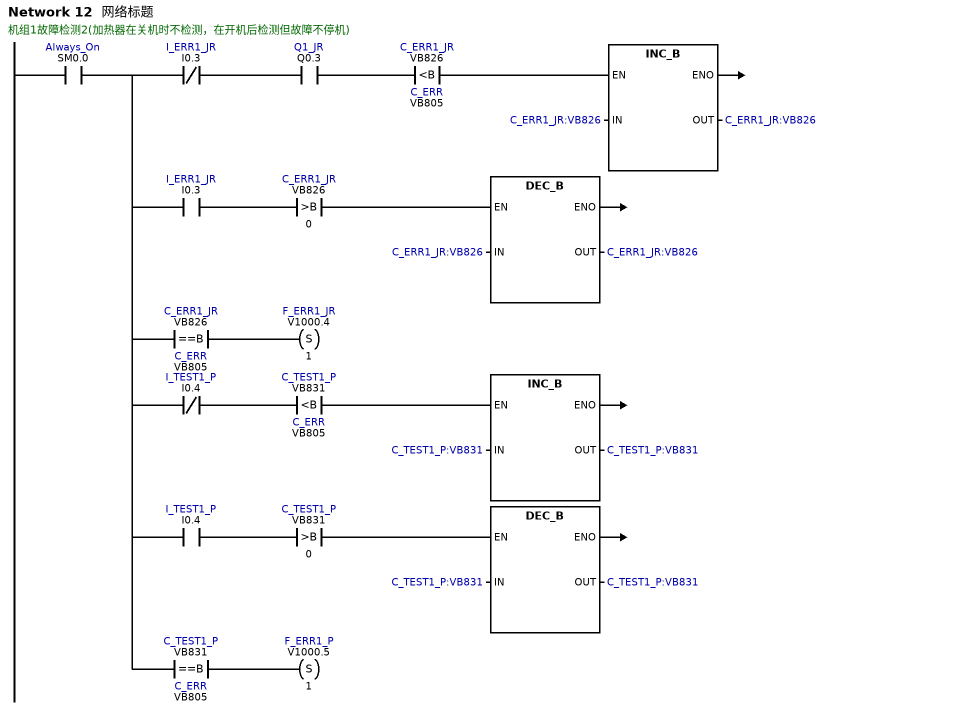
[picture p24: SBR3 networks 12-12]
Network 12 // 网络标题
// 机组1故障检测2(加热器在关机时不检测，在开机后检测但故障不停机)
LD     Always_On:SM0.0
LPS
AN     I_ERR1_JR:I0.3
A      Q1_JR:Q0.3
AB<    C_ERR1_JR:VB826, C_ERR:VB805
INCB   C_ERR1_JR:VB826
LRD
A      I_ERR1_JR:I0.3
AB>    C_ERR1_JR:VB826, 0
DECB   C_ERR1_JR:VB826
LRD
AB=    C_ERR1_JR:VB826, C_ERR:VB805
S      F_ERR1_JR:V1000.4, 1
LRD
AN     I_TEST1_P:I0.4
AB<    C_TEST1_P:VB831, C_ERR:VB805
INCB   C_TEST1_P:VB831
LRD
A      I_TEST1_P:I0.4
AB>    C_TEST1_P:VB831, 0
DECB   C_TEST1_P:VB831
LPP
AB=    C_TEST1_P:VB831, C_ERR:VB805
S      F_ERR1_P:V1000.5, 1
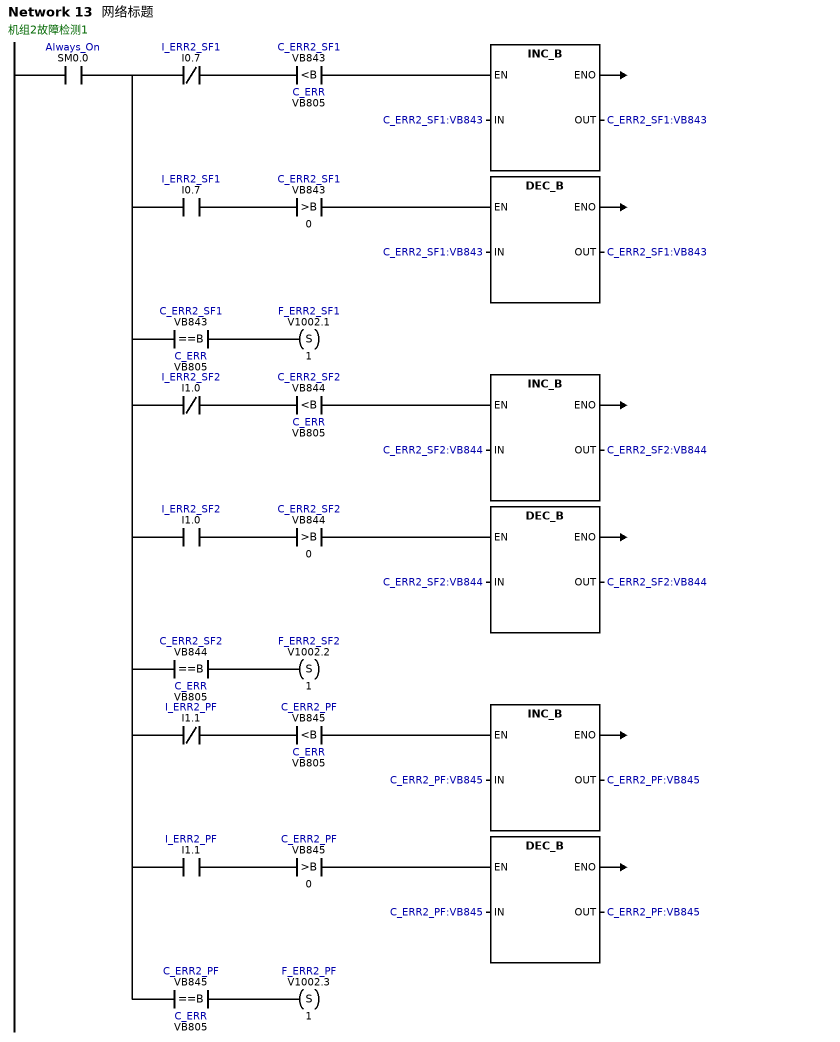
Network 13 // 网络标题
// 机组2故障检测1
LD     Always_On:SM0.0
LPS
AN     I_ERR2_SF1:I0.7
AB<    C_ERR2_SF1:VB843, C_ERR:VB805
INCB   C_ERR2_SF1:VB843
LRD
A      I_ERR2_SF1:I0.7
AB>    C_ERR2_SF1:VB843, 0
DECB   C_ERR2_SF1:VB843
LRD
AB=    C_ERR2_SF1:VB843, C_ERR:VB805
S      F_ERR2_SF1:V1002.1, 1
LRD
AN     I_ERR2_SF2:I1.0
AB<    C_ERR2_SF2:VB844, C_ERR:VB805
INCB   C_ERR2_SF2:VB844
LRD
A      I_ERR2_SF2:I1.0
AB>    C_ERR2_SF2:VB844, 0
DECB   C_ERR2_SF2:VB844
LRD
AB=    C_ERR2_SF2:VB844, C_ERR:VB805
S      F_ERR2_SF2:V1002.2, 1
LRD
AN     I_ERR2_PF:I1.1
AB<    C_ERR2_PF:VB845, C_ERR:VB805
INCB   C_ERR2_PF:VB845
LRD
A      I_ERR2_PF:I1.1
AB>    C_ERR2_PF:VB845, 0
DECB   C_ERR2_PF:VB845
LPP
AB=    C_ERR2_PF:VB845, C_ERR:VB805
S      F_ERR2_PF:V1002.3, 1
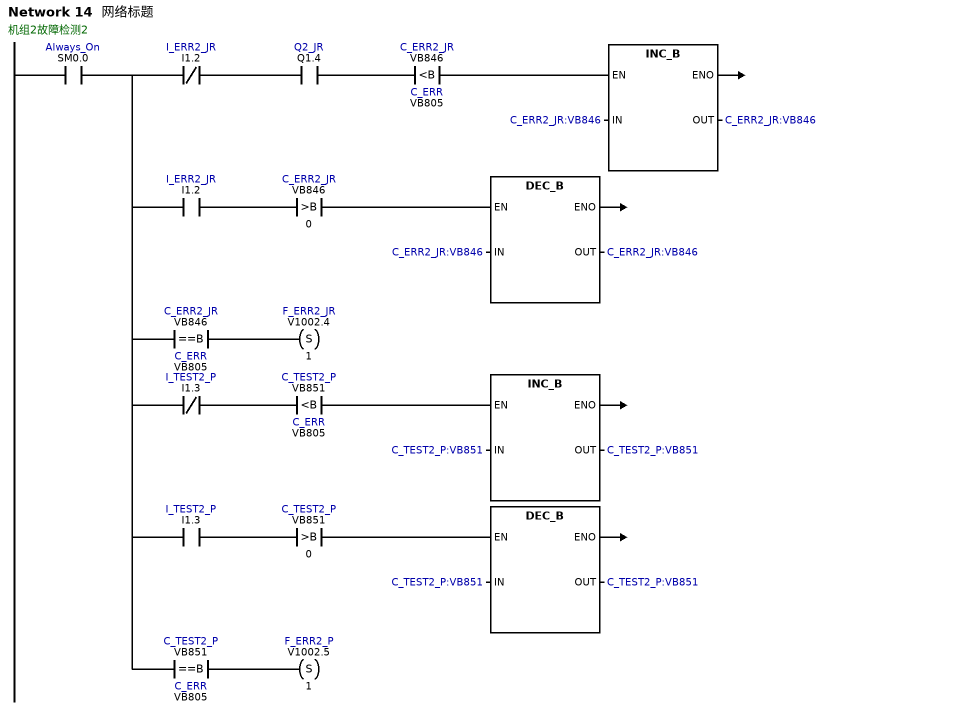
Network 14 // 网络标题
// 机组2故障检测2
LD     Always_On:SM0.0
LPS
AN     I_ERR2_JR:I1.2
A      Q2_JR:Q1.4
AB<    C_ERR2_JR:VB846, C_ERR:VB805
INCB   C_ERR2_JR:VB846
LRD
A      I_ERR2_JR:I1.2
AB>    C_ERR2_JR:VB846, 0
DECB   C_ERR2_JR:VB846
LRD
AB=    C_ERR2_JR:VB846, C_ERR:VB805
S      F_ERR2_JR:V1002.4, 1
LRD
AN     I_TEST2_P:I1.3
AB<    C_TEST2_P:VB851, C_ERR:VB805
INCB   C_TEST2_P:VB851
LRD
A      I_TEST2_P:I1.3
AB>    C_TEST2_P:VB851, 0
DECB   C_TEST2_P:VB851
LPP
AB=    C_TEST2_P:VB851, C_ERR:VB805
S      F_ERR2_P:V1002.5, 1
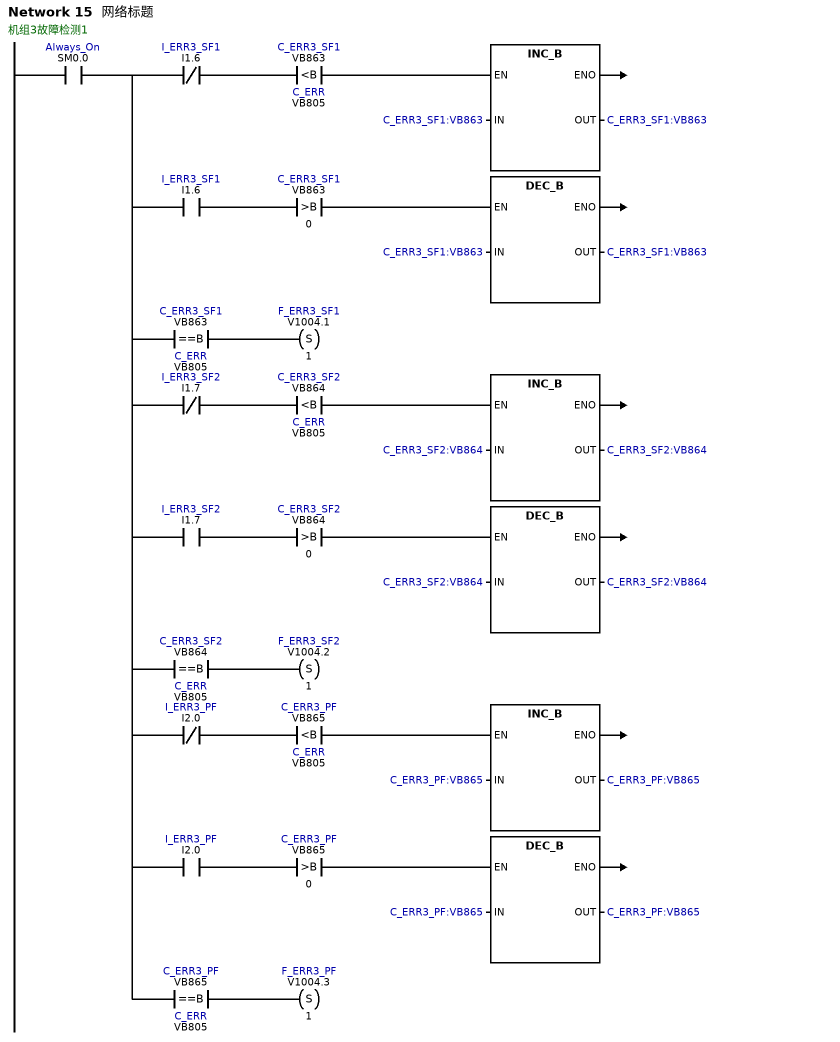
Network 15 // 网络标题
// 机组3故障检测1
LD     Always_On:SM0.0
LPS
AN     I_ERR3_SF1:I1.6
AB<    C_ERR3_SF1:VB863, C_ERR:VB805
INCB   C_ERR3_SF1:VB863
LRD
A      I_ERR3_SF1:I1.6
AB>    C_ERR3_SF1:VB863, 0
DECB   C_ERR3_SF1:VB863
LRD
AB=    C_ERR3_SF1:VB863, C_ERR:VB805
S      F_ERR3_SF1:V1004.1, 1
LRD
AN     I_ERR3_SF2:I1.7
AB<    C_ERR3_SF2:VB864, C_ERR:VB805
INCB   C_ERR3_SF2:VB864
LRD
A      I_ERR3_SF2:I1.7
AB>    C_ERR3_SF2:VB864, 0
DECB   C_ERR3_SF2:VB864
LRD
AB=    C_ERR3_SF2:VB864, C_ERR:VB805
S      F_ERR3_SF2:V1004.2, 1
LRD
AN     I_ERR3_PF:I2.0
AB<    C_ERR3_PF:VB865, C_ERR:VB805
INCB   C_ERR3_PF:VB865
LRD
A      I_ERR3_PF:I2.0
AB>    C_ERR3_PF:VB865, 0
DECB   C_ERR3_PF:VB865
LPP
AB=    C_ERR3_PF:VB865, C_ERR:VB805
S      F_ERR3_PF:V1004.3, 1
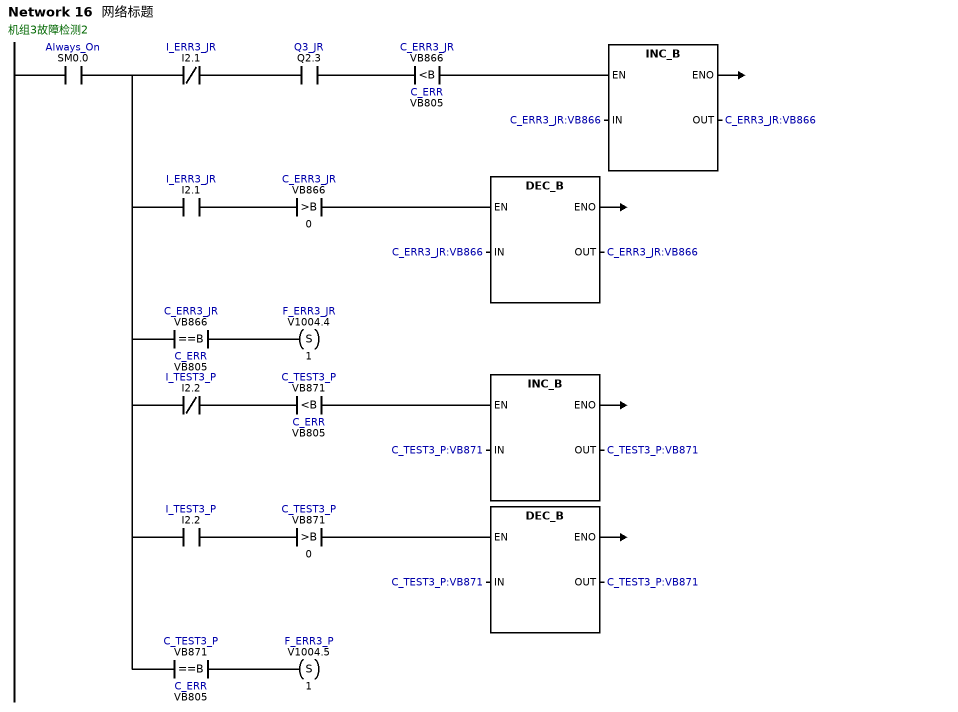
Network 16 // 网络标题
// 机组3故障检测2
LD     Always_On:SM0.0
LPS
AN     I_ERR3_JR:I2.1
A      Q3_JR:Q2.3
AB<    C_ERR3_JR:VB866, C_ERR:VB805
INCB   C_ERR3_JR:VB866
LRD
A      I_ERR3_JR:I2.1
AB>    C_ERR3_JR:VB866, 0
DECB   C_ERR3_JR:VB866
LRD
AB=    C_ERR3_JR:VB866, C_ERR:VB805
S      F_ERR3_JR:V1004.4, 1
LRD
AN     I_TEST3_P:I2.2
AB<    C_TEST3_P:VB871, C_ERR:VB805
INCB   C_TEST3_P:VB871
LRD
A      I_TEST3_P:I2.2
AB>    C_TEST3_P:VB871, 0
DECB   C_TEST3_P:VB871
LPP
AB=    C_TEST3_P:VB871, C_ERR:VB805
S      F_ERR3_P:V1004.5, 1
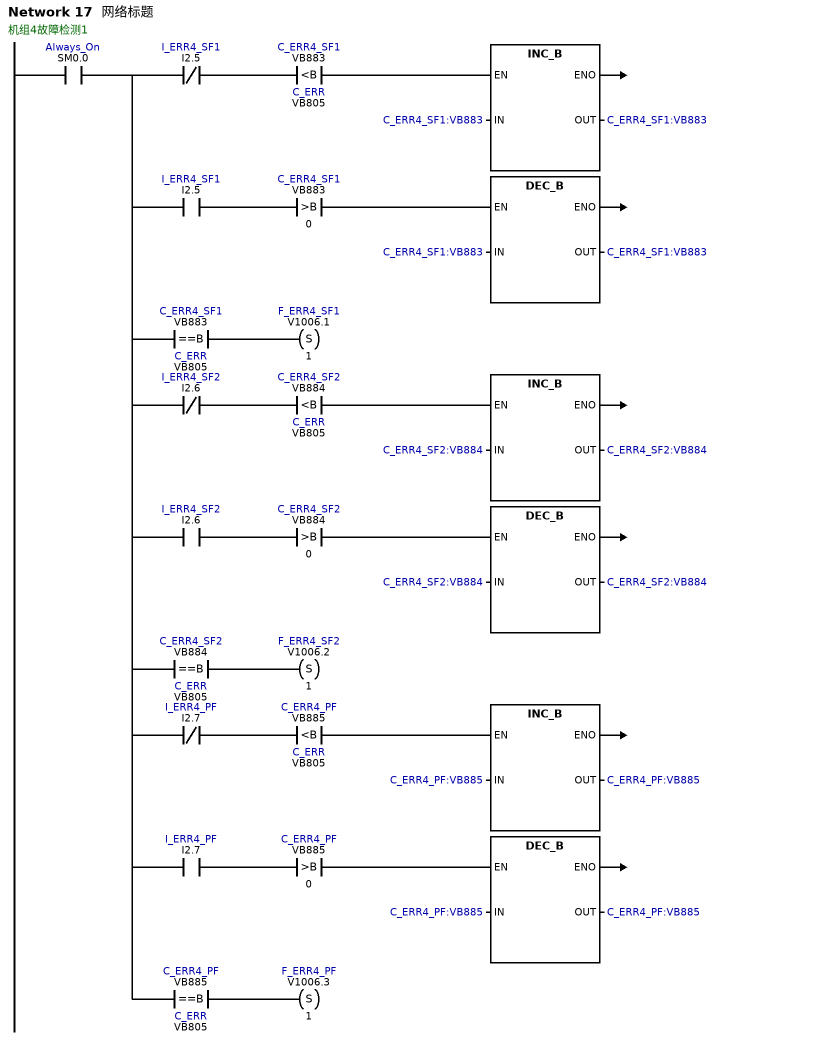
Network 17 // 网络标题
// 机组4故障检测1
LD     Always_On:SM0.0
LPS
AN     I_ERR4_SF1:I2.5
AB<    C_ERR4_SF1:VB883, C_ERR:VB805
INCB   C_ERR4_SF1:VB883
LRD
A      I_ERR4_SF1:I2.5
AB>    C_ERR4_SF1:VB883, 0
DECB   C_ERR4_SF1:VB883
LRD
AB=    C_ERR4_SF1:VB883, C_ERR:VB805
S      F_ERR4_SF1:V1006.1, 1
LRD
AN     I_ERR4_SF2:I2.6
AB<    C_ERR4_SF2:VB884, C_ERR:VB805
INCB   C_ERR4_SF2:VB884
LRD
A      I_ERR4_SF2:I2.6
AB>    C_ERR4_SF2:VB884, 0
DECB   C_ERR4_SF2:VB884
LRD
AB=    C_ERR4_SF2:VB884, C_ERR:VB805
S      F_ERR4_SF2:V1006.2, 1
LRD
AN     I_ERR4_PF:I2.7
AB<    C_ERR4_PF:VB885, C_ERR:VB805
INCB   C_ERR4_PF:VB885
LRD
A      I_ERR4_PF:I2.7
AB>    C_ERR4_PF:VB885, 0
DECB   C_ERR4_PF:VB885
LPP
AB=    C_ERR4_PF:VB885, C_ERR:VB805
S      F_ERR4_PF:V1006.3, 1
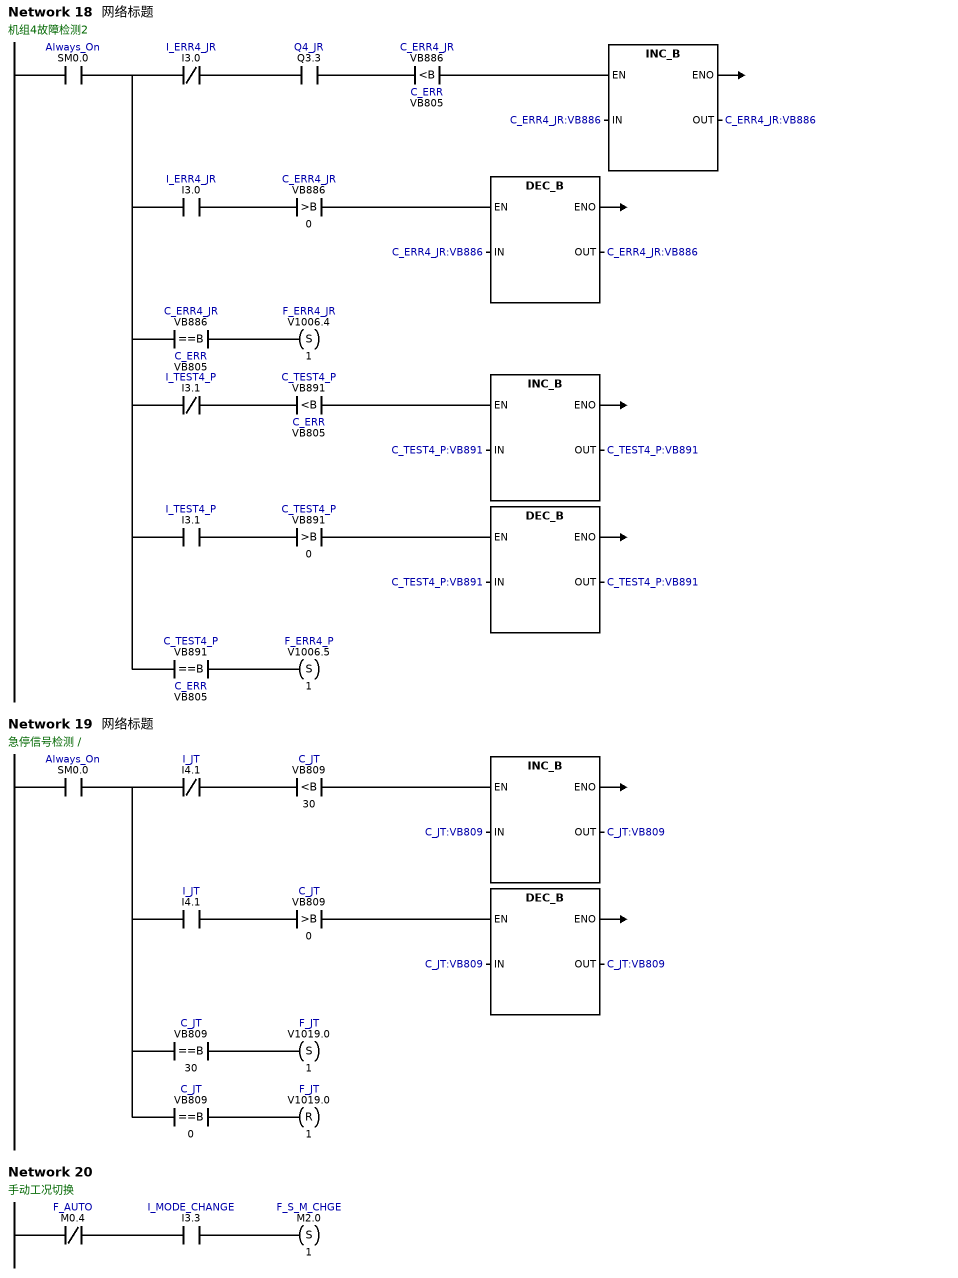
Network 18 // 网络标题
// 机组4故障检测2
LD     Always_On:SM0.0
LPS
AN     I_ERR4_JR:I3.0
A      Q4_JR:Q3.3
AB<    C_ERR4_JR:VB886, C_ERR:VB805
INCB   C_ERR4_JR:VB886
LRD
A      I_ERR4_JR:I3.0
AB>    C_ERR4_JR:VB886, 0
DECB   C_ERR4_JR:VB886
LRD
AB=    C_ERR4_JR:VB886, C_ERR:VB805
S      F_ERR4_JR:V1006.4, 1
LRD
AN     I_TEST4_P:I3.1
AB<    C_TEST4_P:VB891, C_ERR:VB805
INCB   C_TEST4_P:VB891
LRD
A      I_TEST4_P:I3.1
AB>    C_TEST4_P:VB891, 0
DECB   C_TEST4_P:VB891
LPP
AB=    C_TEST4_P:VB891, C_ERR:VB805
S      F_ERR4_P:V1006.5, 1
Network 19 // 网络标题
// 急停信号检测
// 
LD     Always_On:SM0.0
LPS
AN     I_JT:I4.1
AB<    C_JT:VB809, 30
INCB   C_JT:VB809
LRD
A      I_JT:I4.1
AB>    C_JT:VB809, 0
DECB   C_JT:VB809
LRD
AB=    C_JT:VB809, 30
S      F_JT:V1019.0, 1
LPP
AB=    C_JT:VB809, 0
R      F_JT:V1019.0, 1
Network 20
// 手动工况切换
LDN    F_AUTO:M0.4
A      I_MODE_CHANGE:I3.3
S      F_S_M_CHGE:M2.0, 1
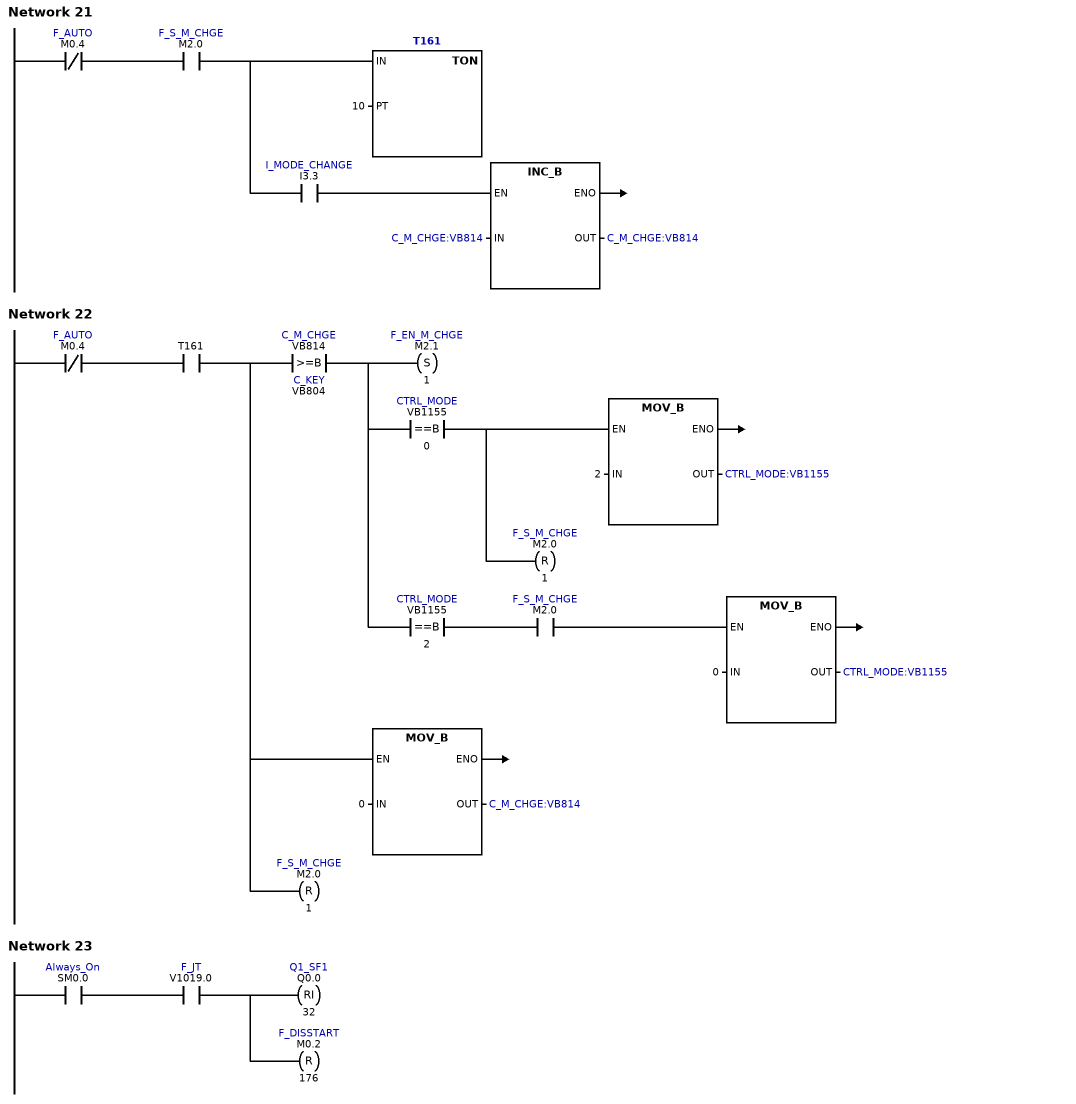
Network 21
LDN    F_AUTO:M0.4
A      F_S_M_CHGE:M2.0
TON    T161, 10
A      I_MODE_CHANGE:I3.3
INCB   C_M_CHGE:VB814
Network 22
LDN    F_AUTO:M0.4
A      T161
LPS
AB>=   C_M_CHGE:VB814, C_KEY:VB804
LPS
S      F_EN_M_CHGE:M2.1, 1
AB=    CTRL_MODE:VB1155, 0
MOVB   2, CTRL_MODE:VB1155
R      F_S_M_CHGE:M2.0, 1
LPP
AB=    CTRL_MODE:VB1155, 2
A      F_S_M_CHGE:M2.0
MOVB   0, CTRL_MODE:VB1155
LPP
MOVB   0, C_M_CHGE:VB814
R      F_S_M_CHGE:M2.0, 1
Network 23
LD     Always_On:SM0.0
A      F_JT:V1019.0
RI     Q1_SF1:Q0.0, 32
R      F_DISSTART:M0.2, 176
END_SUBROUTINE_BLOCK

// SBR4: protected block, not included

SUBROUTINE_BLOCK 参数设定:SBR5
TITLE=
VAR
TEMP_W:WORD;	// LW0 
TEMP_W1:WORD;	// LW2 
TEMP_W2:WORD;	// LW4 
END_VAR
BEGIN
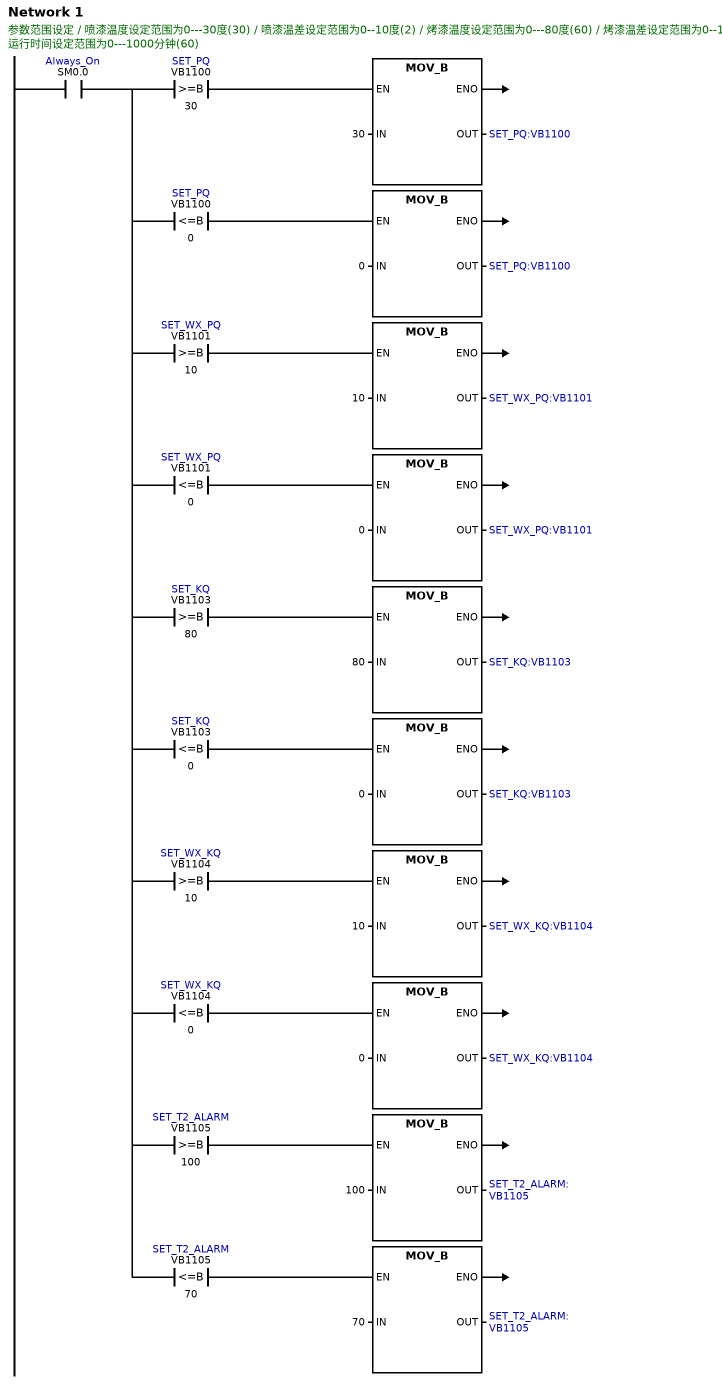
Network 1
// 参数范围设定
// 喷漆温度设定范围为0---30度(30)
// 喷漆温差设定范围为0--10度(2)
// 烤漆温度设定范围为0---80度(60)
// 烤漆温差设定范围为0--10度(2)
// T2超温保护温度设定范围为70---100度(85)
// 运行时间设定范围为0---1000分钟(60)
LD     Always_On:SM0.0
LPS
AB>=   SET_PQ:VB1100, 30
MOVB   30, SET_PQ:VB1100
LRD
AB<=   SET_PQ:VB1100, 0
MOVB   0, SET_PQ:VB1100
LRD
AB>=   SET_WX_PQ:VB1101, 10
MOVB   10, SET_WX_PQ:VB1101
LRD
AB<=   SET_WX_PQ:VB1101, 0
MOVB   0, SET_WX_PQ:VB1101
LRD
AB>=   SET_KQ:VB1103, 80
MOVB   80, SET_KQ:VB1103
LRD
AB<=   SET_KQ:VB1103, 0
MOVB   0, SET_KQ:VB1103
LRD
AB>=   SET_WX_KQ:VB1104, 10
MOVB   10, SET_WX_KQ:VB1104
LRD
AB<=   SET_WX_KQ:VB1104, 0
MOVB   0, SET_WX_KQ:VB1104
LRD
AB>=   SET_T2_ALARM:VB1105, 100
MOVB   100, SET_T2_ALARM:VB1105
LPP
AB<=   SET_T2_ALARM:VB1105, 70
MOVB   70, SET_T2_ALARM:VB1105
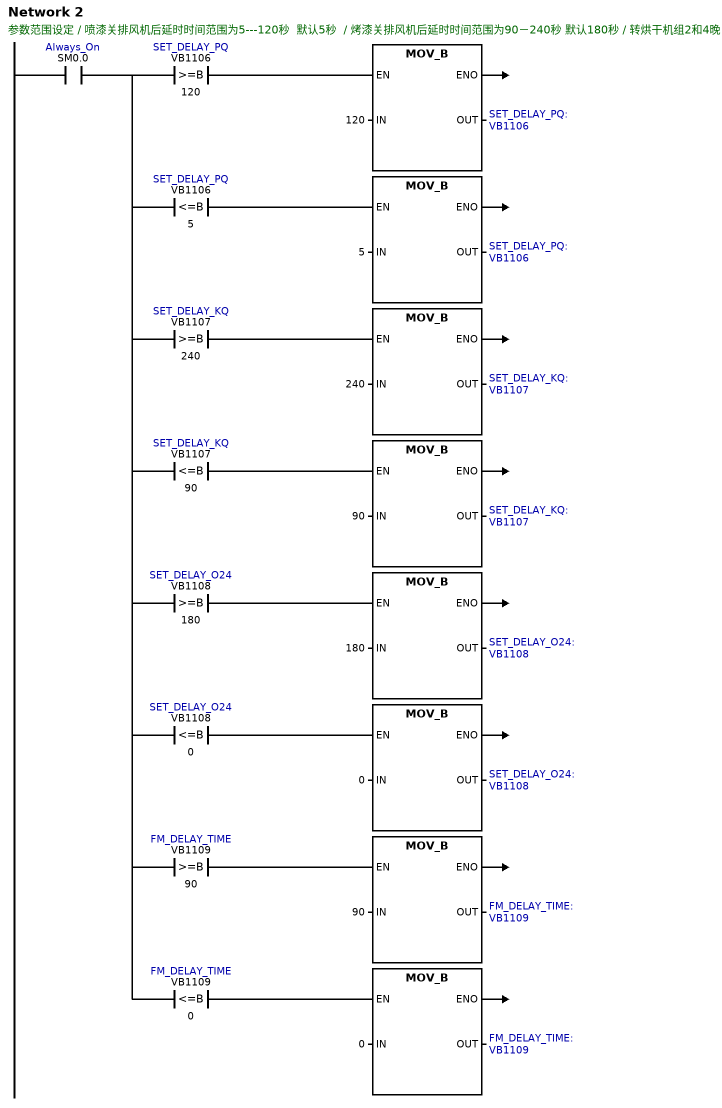
Network 2
// 参数范围设定
// 喷漆关排风机后延时时间范围为5---120秒  默认5秒 
// 烤漆关排风机后延时时间范围为90－240秒 默认180秒
// 转烘干机组2和4晚关延时时间为0－180秒   默认30秒
LD     Always_On:SM0.0
LPS
AB>=   SET_DELAY_PQ:VB1106, 120
MOVB   120, SET_DELAY_PQ:VB1106
LRD
AB<=   SET_DELAY_PQ:VB1106, 5
MOVB   5, SET_DELAY_PQ:VB1106
LRD
AB>=   SET_DELAY_KQ:VB1107, 240
MOVB   240, SET_DELAY_KQ:VB1107
LRD
AB<=   SET_DELAY_KQ:VB1107, 90
MOVB   90, SET_DELAY_KQ:VB1107
LRD
AB>=   SET_DELAY_O24:VB1108, 180
MOVB   180, SET_DELAY_O24:VB1108
LRD
AB<=   SET_DELAY_O24:VB1108, 0
MOVB   0, SET_DELAY_O24:VB1108
LRD
AB>=   FM_DELAY_TIME:VB1109, 90
MOVB   90, FM_DELAY_TIME:VB1109
LPP
AB<=   FM_DELAY_TIME:VB1109, 0
MOVB   0, FM_DELAY_TIME:VB1109
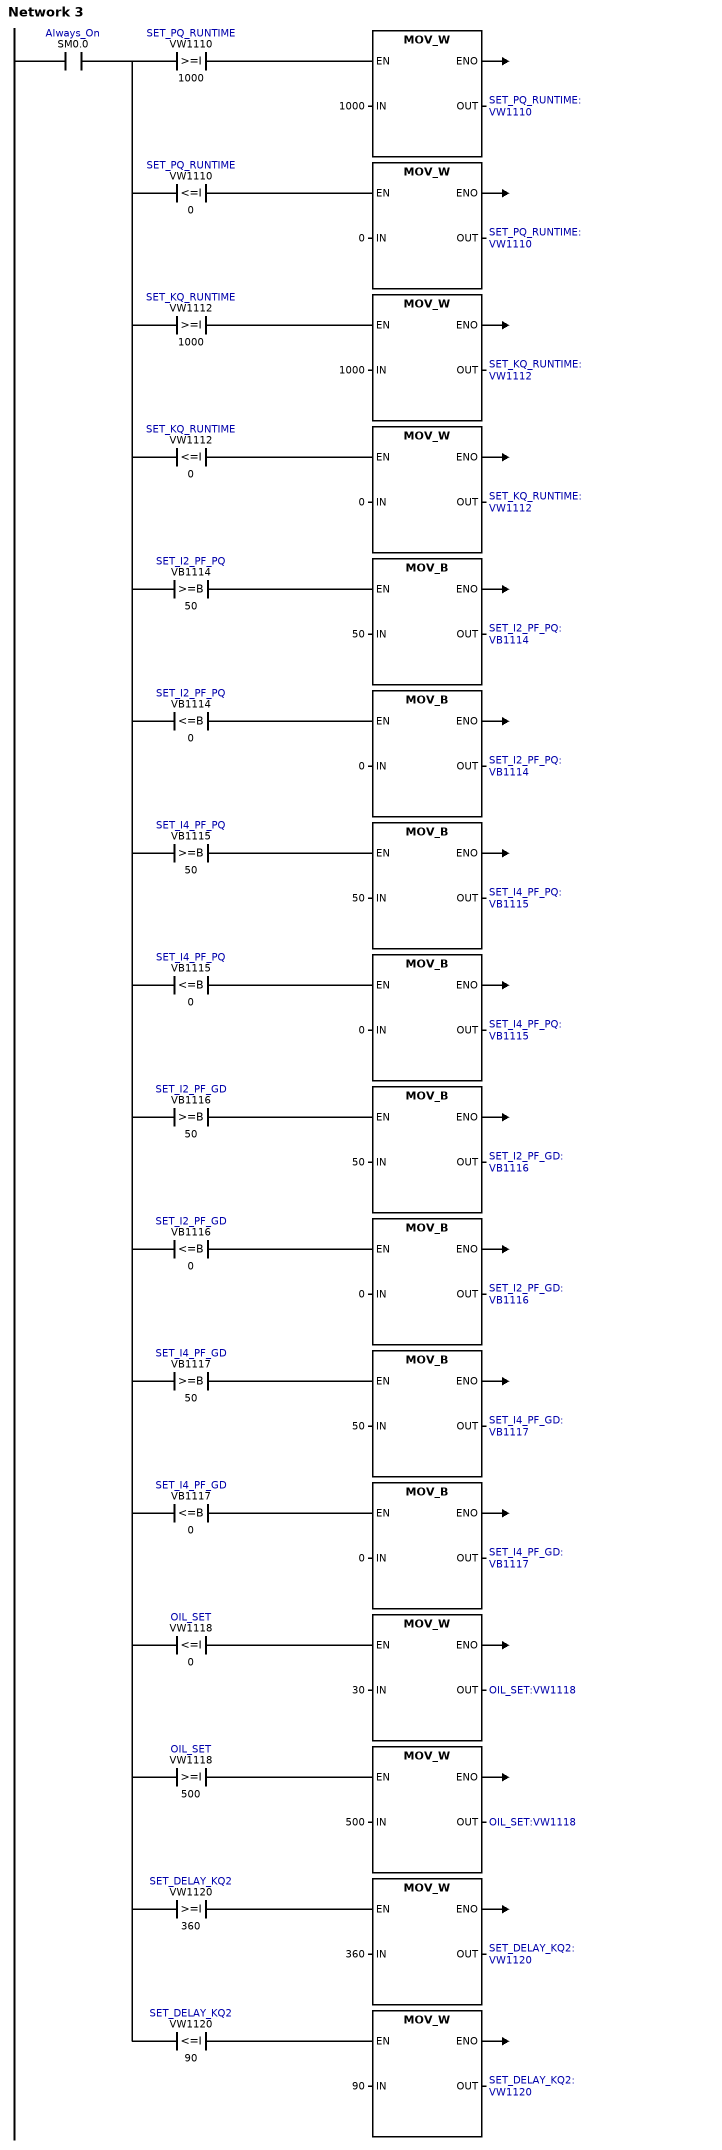
Network 3
LD     Always_On:SM0.0
LPS
AW>=   SET_PQ_RUNTIME:VW1110, 1000
MOVW   1000, SET_PQ_RUNTIME:VW1110
LRD
AW<=   SET_PQ_RUNTIME:VW1110, 0
MOVW   0, SET_PQ_RUNTIME:VW1110
LRD
AW>=   SET_KQ_RUNTIME:VW1112, 1000
MOVW   1000, SET_KQ_RUNTIME:VW1112
LRD
AW<=   SET_KQ_RUNTIME:VW1112, 0
MOVW   0, SET_KQ_RUNTIME:VW1112
LRD
AB>=   SET_I2_PF_PQ:VB1114, 50
MOVB   50, SET_I2_PF_PQ:VB1114
LRD
AB<=   SET_I2_PF_PQ:VB1114, 0
MOVB   0, SET_I2_PF_PQ:VB1114
LRD
AB>=   SET_I4_PF_PQ:VB1115, 50
MOVB   50, SET_I4_PF_PQ:VB1115
LRD
AB<=   SET_I4_PF_PQ:VB1115, 0
MOVB   0, SET_I4_PF_PQ:VB1115
LRD
AB>=   SET_I2_PF_GD:VB1116, 50
MOVB   50, SET_I2_PF_GD:VB1116
LRD
AB<=   SET_I2_PF_GD:VB1116, 0
MOVB   0, SET_I2_PF_GD:VB1116
LRD
AB>=   SET_I4_PF_GD:VB1117, 50
MOVB   50, SET_I4_PF_GD:VB1117
LRD
AB<=   SET_I4_PF_GD:VB1117, 0
MOVB   0, SET_I4_PF_GD:VB1117
LRD
AW<=   OIL_SET:VW1118, 0
MOVW   30, OIL_SET:VW1118
LRD
AW>=   OIL_SET:VW1118, 500
MOVW   500, OIL_SET:VW1118
LRD
AW>=   SET_DELAY_KQ2:VW1120, 360
MOVW   360, SET_DELAY_KQ2:VW1120
LPP
AW<=   SET_DELAY_KQ2:VW1120, 90
MOVW   90, SET_DELAY_KQ2:VW1120
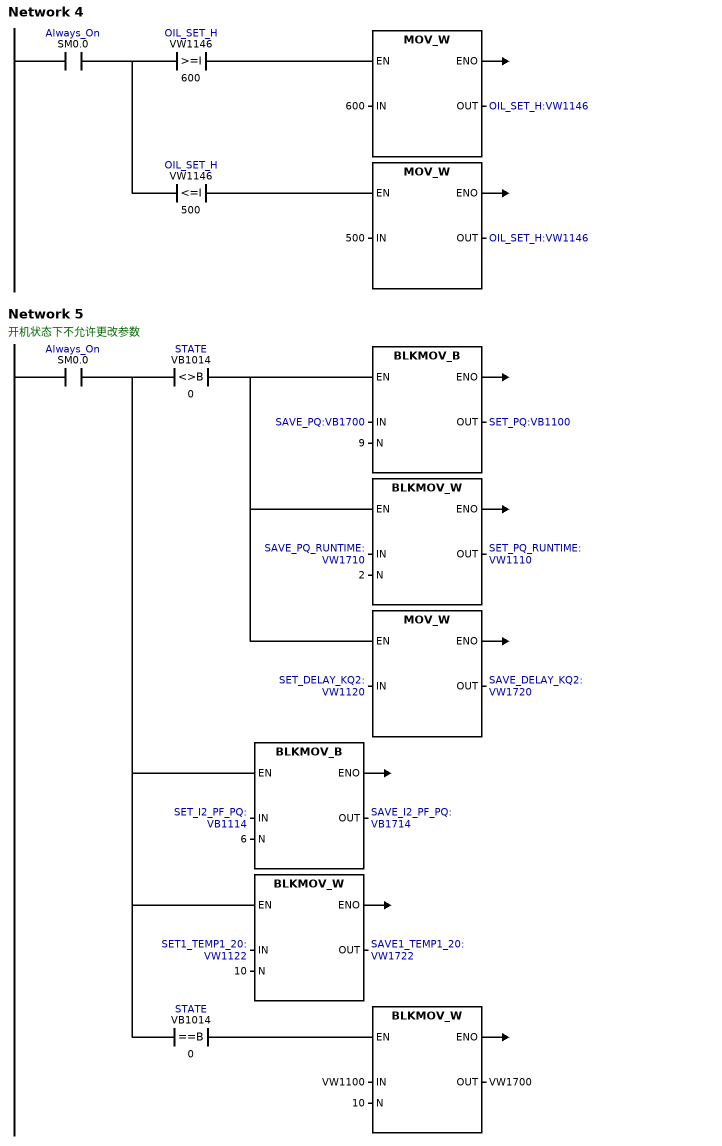
Network 4
LD     Always_On:SM0.0
LPS
AW>=   OIL_SET_H:VW1146, 600
MOVW   600, OIL_SET_H:VW1146
LPP
AW<=   OIL_SET_H:VW1146, 500
MOVW   500, OIL_SET_H:VW1146
Network 5
// 开机状态下不允许更改参数
LD     Always_On:SM0.0
LPS
AB<>   STATE:VB1014, 0
BMB    SAVE_PQ:VB1700, SET_PQ:VB1100, 9
BMW    SAVE_PQ_RUNTIME:VW1710, SET_PQ_RUNTIME:VW1110, 2
MOVW   SET_DELAY_KQ2:VW1120, SAVE_DELAY_KQ2:VW1720
LPP
BMB    SET_I2_PF_PQ:VB1114, SAVE_I2_PF_PQ:VB1714, 6
BMW    SET1_TEMP1_20:VW1122, SAVE1_TEMP1_20:VW1722, 10
AB=    STATE:VB1014, 0
BMW    VW1100, VW1700, 10
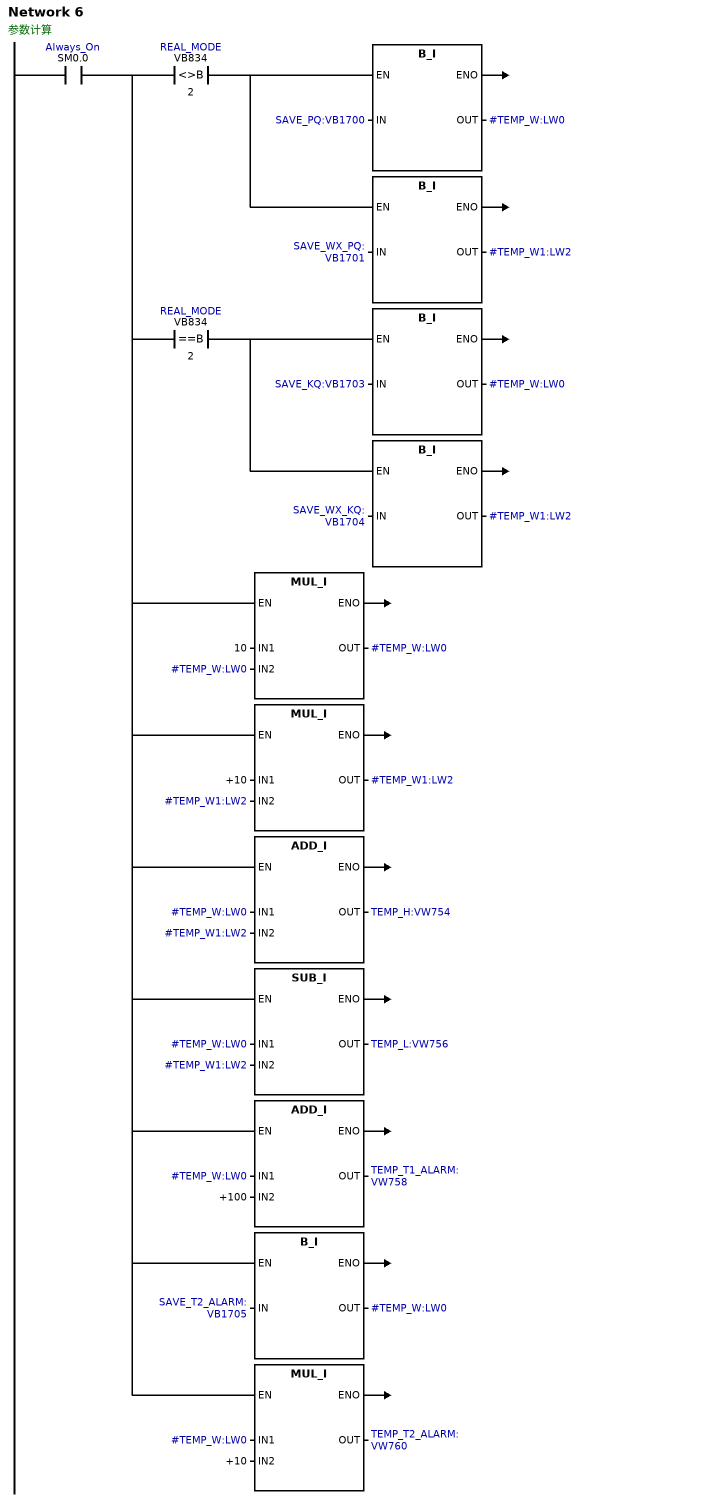
Network 6
// 参数计算
LD     Always_On:SM0.0
LPS
AB<>   REAL_MODE:VB834, 2
BTI    SAVE_PQ:VB1700, #TEMP_W:LW0
BTI    SAVE_WX_PQ:VB1701, #TEMP_W1:LW2
LRD
AB=    REAL_MODE:VB834, 2
BTI    SAVE_KQ:VB1703, #TEMP_W:LW0
BTI    SAVE_WX_KQ:VB1704, #TEMP_W1:LW2
LPP
*I     10, #TEMP_W:LW0
*I     +10, #TEMP_W1:LW2
MOVW   #TEMP_W:LW0, TEMP_H:VW754
+I     #TEMP_W1:LW2, TEMP_H:VW754
MOVW   #TEMP_W:LW0, TEMP_L:VW756
-I     #TEMP_W1:LW2, TEMP_L:VW756
MOVW   #TEMP_W:LW0, TEMP_T1_ALARM:VW758
+I     +100, TEMP_T1_ALARM:VW758
BTI    SAVE_T2_ALARM:VB1705, #TEMP_W:LW0
MOVW   #TEMP_W:LW0, TEMP_T2_ALARM:VW760
*I     +10, TEMP_T2_ALARM:VW760
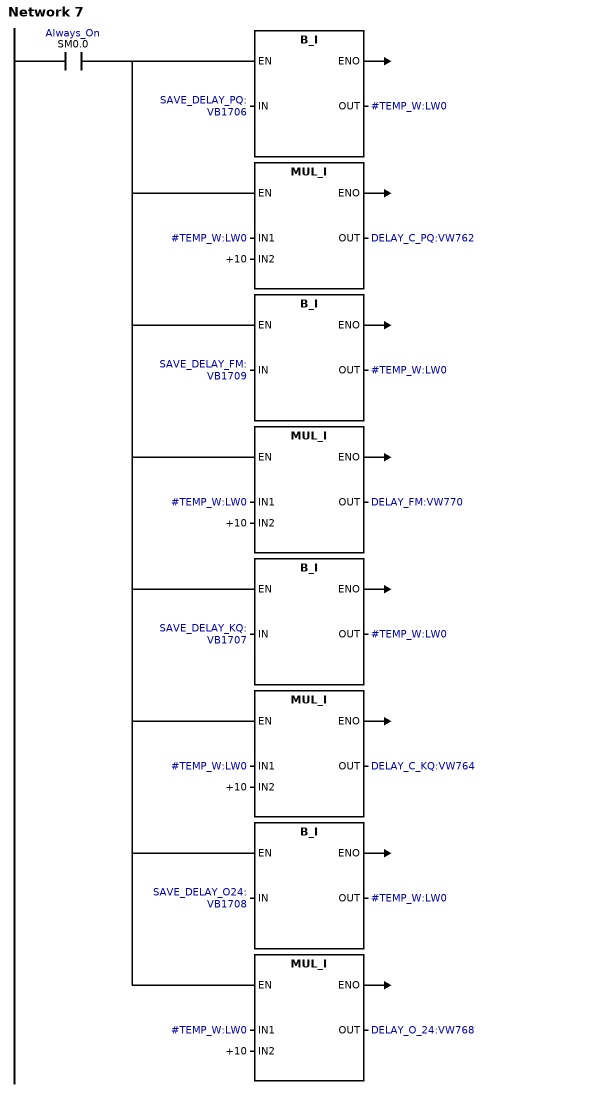
Network 7
LD     Always_On:SM0.0
BTI    SAVE_DELAY_PQ:VB1706, #TEMP_W:LW0
MOVW   #TEMP_W:LW0, DELAY_C_PQ:VW762
*I     +10, DELAY_C_PQ:VW762
BTI    SAVE_DELAY_FM:VB1709, #TEMP_W:LW0
MOVW   #TEMP_W:LW0, DELAY_FM:VW770
*I     +10, DELAY_FM:VW770
BTI    SAVE_DELAY_KQ:VB1707, #TEMP_W:LW0
MOVW   #TEMP_W:LW0, DELAY_C_KQ:VW764
*I     +10, DELAY_C_KQ:VW764
BTI    SAVE_DELAY_O24:VB1708, #TEMP_W:LW0
MOVW   #TEMP_W:LW0, DELAY_O_24:VW768
*I     +10, DELAY_O_24:VW768
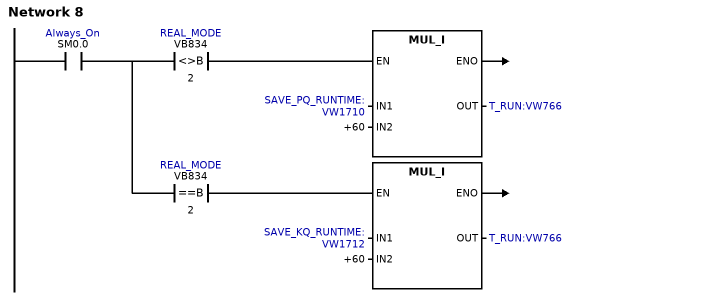
Network 8
LD     Always_On:SM0.0
LPS
AB<>   REAL_MODE:VB834, 2
MOVW   SAVE_PQ_RUNTIME:VW1710, T_RUN:VW766
*I     +60, T_RUN:VW766
LPP
AB=    REAL_MODE:VB834, 2
MOVW   SAVE_KQ_RUNTIME:VW1712, T_RUN:VW766
*I     +60, T_RUN:VW766
END_SUBROUTINE_BLOCK

SUBROUTINE_BLOCK 温度采样:SBR6
TITLE=
VAR_INPUT
ADDRESS:DWORD;	// LD0 
IN:WORD;	// LW4 
IN_TEMP:WORD;	// LW6 
F_SET:BOOL;	// L8.0 
END_VAR
VAR_OUTPUT
OUT:WORD;	// LW9 
AVERAGE:WORD;	// LW11 
OUT_TEMP:WORD;	// LW13 
END_VAR
VAR
MAX:WORD;	// LW15 
MIN:WORD;	// LW17 
TEMP_B:BYTE;	// LB19 
TEMP_W:WORD;	// LW20 
TEMP_DW:DWORD;	// LD22 
SUM:DWORD;	// LD26 
PP1:DWORD;	// LD30 
PP2:DWORD;	// LD34 
TEMP_W2:WORD;	// LW38 
AC_TEMP:DWORD;	// LD40 
END_VAR
BEGIN
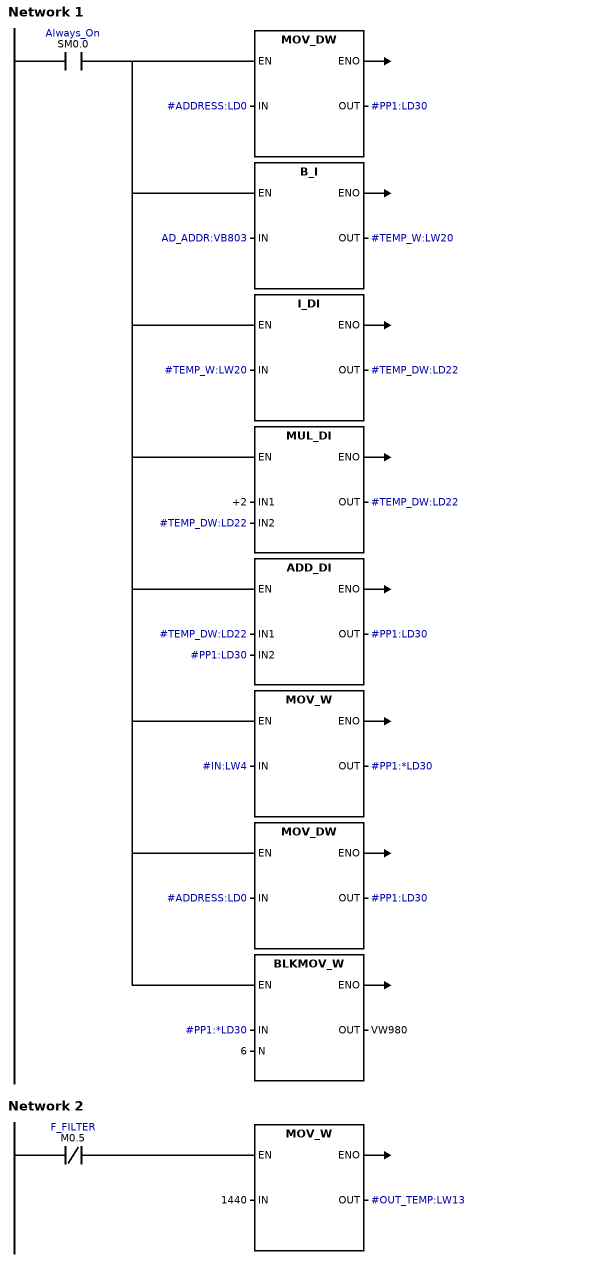
Network 1
LD     Always_On:SM0.0
MOVD   #ADDRESS:LD0, #PP1:LD30
BTI    AD_ADDR:VB803, #TEMP_W:LW20
ITD    #TEMP_W:LW20, #TEMP_DW:LD22
*D     +2, #TEMP_DW:LD22
+D     #TEMP_DW:LD22, #PP1:LD30
MOVW   #IN:LW4, *#PP1:LD30
MOVD   #ADDRESS:LD0, #PP1:LD30
BMW    *#PP1:LD30, VW980, 6
Network 2
LDN    F_FILTER:M0.5
MOVW   1440, #OUT_TEMP:LW13
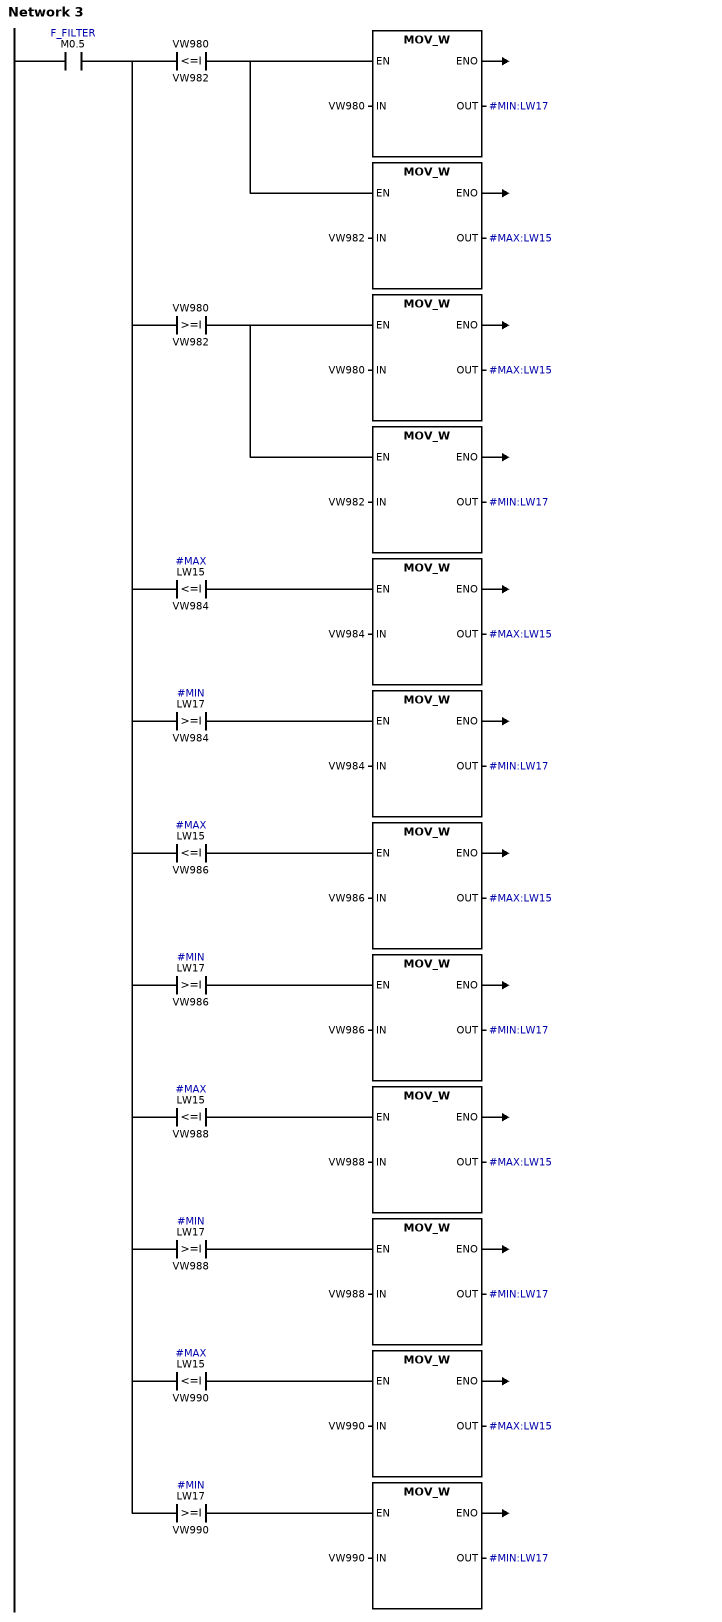
Network 3
LD     F_FILTER:M0.5
LPS
AW<=   VW980, VW982
MOVW   VW980, #MIN:LW17
MOVW   VW982, #MAX:LW15
LRD
AW>=   VW980, VW982
MOVW   VW980, #MAX:LW15
MOVW   VW982, #MIN:LW17
LPP
LPS
AW<=   #MAX:LW15, VW984
MOVW   VW984, #MAX:LW15
LRD
AW>=   #MIN:LW17, VW984
MOVW   VW984, #MIN:LW17
LRD
AW<=   #MAX:LW15, VW986
MOVW   VW986, #MAX:LW15
LRD
AW>=   #MIN:LW17, VW986
MOVW   VW986, #MIN:LW17
LRD
AW<=   #MAX:LW15, VW988
MOVW   VW988, #MAX:LW15
LRD
AW>=   #MIN:LW17, VW988
MOVW   VW988, #MIN:LW17
LRD
AW<=   #MAX:LW15, VW990
MOVW   VW990, #MAX:LW15
LPP
AW>=   #MIN:LW17, VW990
MOVW   VW990, #MIN:LW17
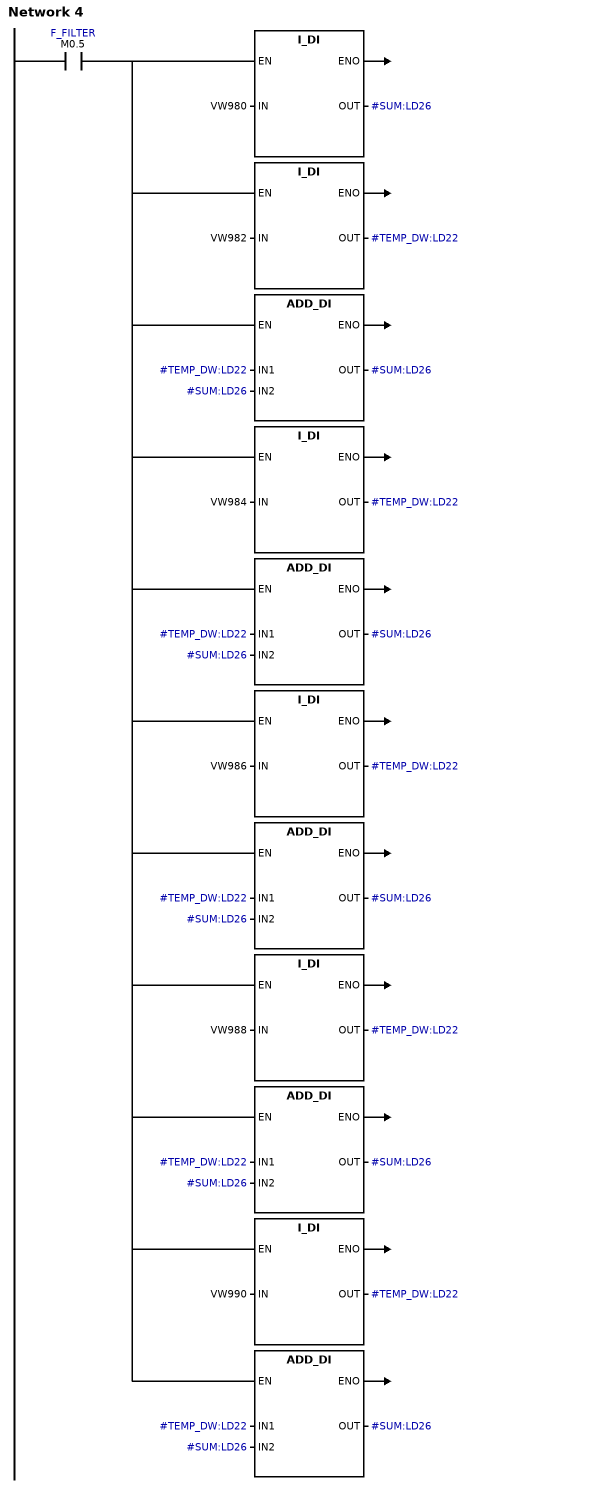
Network 4
LD     F_FILTER:M0.5
ITD    VW980, #SUM:LD26
ITD    VW982, #TEMP_DW:LD22
+D     #TEMP_DW:LD22, #SUM:LD26
ITD    VW984, #TEMP_DW:LD22
+D     #TEMP_DW:LD22, #SUM:LD26
ITD    VW986, #TEMP_DW:LD22
+D     #TEMP_DW:LD22, #SUM:LD26
ITD    VW988, #TEMP_DW:LD22
+D     #TEMP_DW:LD22, #SUM:LD26
ITD    VW990, #TEMP_DW:LD22
+D     #TEMP_DW:LD22, #SUM:LD26
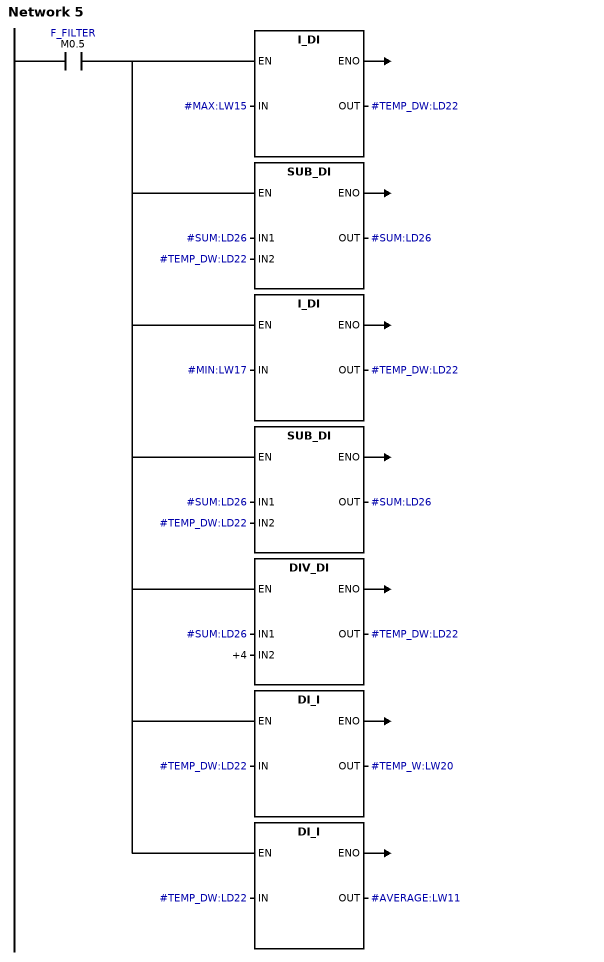
Network 5
LD     F_FILTER:M0.5
ITD    #MAX:LW15, #TEMP_DW:LD22
-D     #TEMP_DW:LD22, #SUM:LD26
ITD    #MIN:LW17, #TEMP_DW:LD22
-D     #TEMP_DW:LD22, #SUM:LD26
MOVD   #SUM:LD26, #TEMP_DW:LD22
/D     +4, #TEMP_DW:LD22
DTI    #TEMP_DW:LD22, #TEMP_W:LW20
DTI    #TEMP_DW:LD22, #AVERAGE:LW11
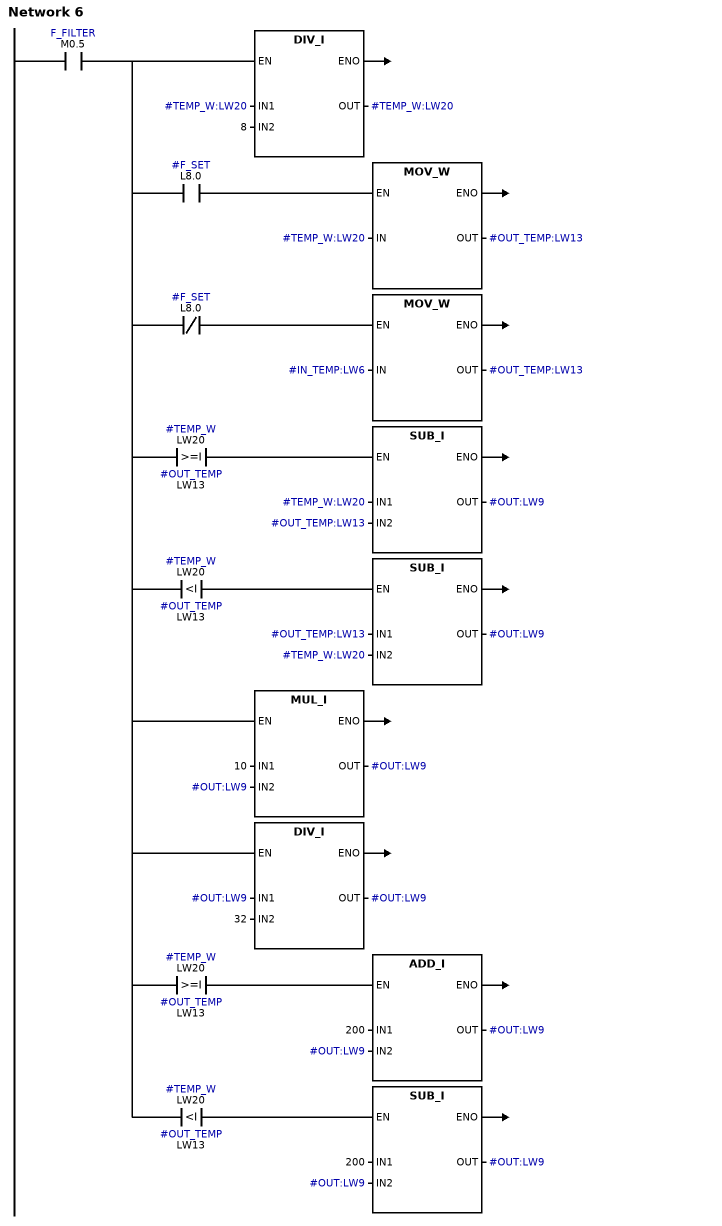
Network 6
LD     F_FILTER:M0.5
LPS
/I     8, #TEMP_W:LW20
A      #F_SET:L8.0
MOVW   #TEMP_W:LW20, #OUT_TEMP:LW13
LRD
AN     #F_SET:L8.0
MOVW   #IN_TEMP:LW6, #OUT_TEMP:LW13
LRD
AW>=   #TEMP_W:LW20, #OUT_TEMP:LW13
MOVW   #TEMP_W:LW20, #OUT:LW9
-I     #OUT_TEMP:LW13, #OUT:LW9
LRD
AW<    #TEMP_W:LW20, #OUT_TEMP:LW13
MOVW   #OUT_TEMP:LW13, #OUT:LW9
-I     #TEMP_W:LW20, #OUT:LW9
LRD
*I     10, #OUT:LW9
LRD
/I     32, #OUT:LW9
LRD
AW>=   #TEMP_W:LW20, #OUT_TEMP:LW13
+I     200, #OUT:LW9
LPP
AW<    #TEMP_W:LW20, #OUT_TEMP:LW13
INVW   #OUT:LW9
INCW   #OUT:LW9
+I     200, #OUT:LW9
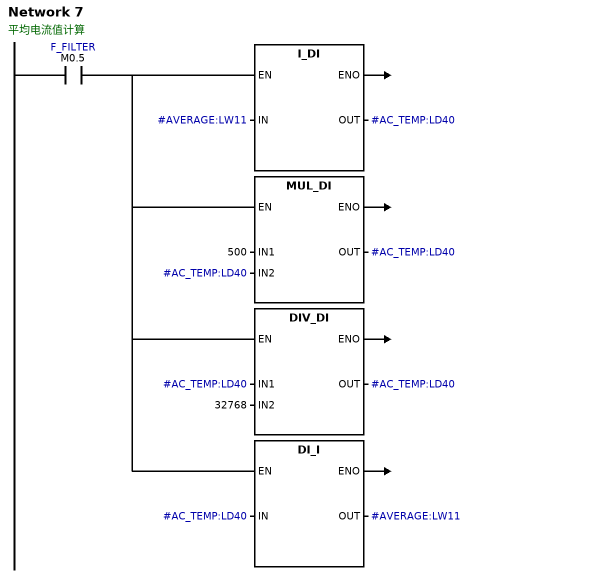
Network 7
// 平均电流值计算
LD     F_FILTER:M0.5
ITD    #AVERAGE:LW11, #AC_TEMP:LD40
*D     500, #AC_TEMP:LD40
/D     32768, #AC_TEMP:LD40
DTI    #AC_TEMP:LD40, #AVERAGE:LW11
END_SUBROUTINE_BLOCK

SUBROUTINE_BLOCK 启动停止控制:SBR7
TITLE=
BEGIN
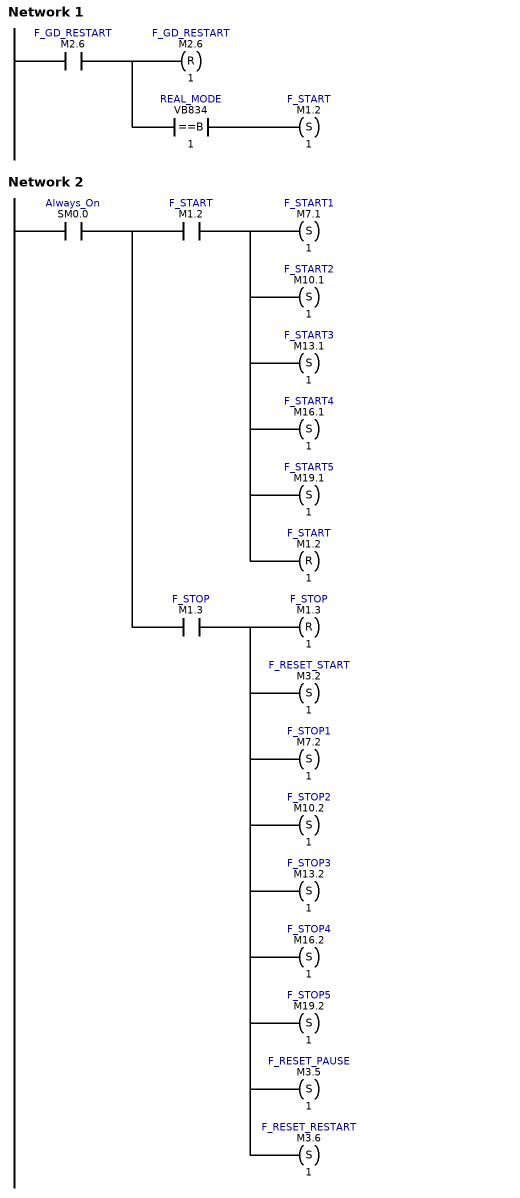
Network 1
LD     F_GD_RESTART:M2.6
R      F_GD_RESTART:M2.6, 1
AB=    REAL_MODE:VB834, 1
S      F_START:M1.2, 1
Network 2
LD     Always_On:SM0.0
LPS
A      F_START:M1.2
S      F_START1:M7.1, 1
S      F_START2:M10.1, 1
S      F_START3:M13.1, 1
S      F_START4:M16.1, 1
S      F_START5:M19.1, 1
R      F_START:M1.2, 1
LPP
A      F_STOP:M1.3
R      F_STOP:M1.3, 1
S      F_RESET_START:M3.2, 1
S      F_STOP1:M7.2, 1
S      F_STOP2:M10.2, 1
S      F_STOP3:M13.2, 1
S      F_STOP4:M16.2, 1
S      F_STOP5:M19.2, 1
S      F_RESET_PAUSE:M3.5, 1
S      F_RESET_RESTART:M3.6, 1
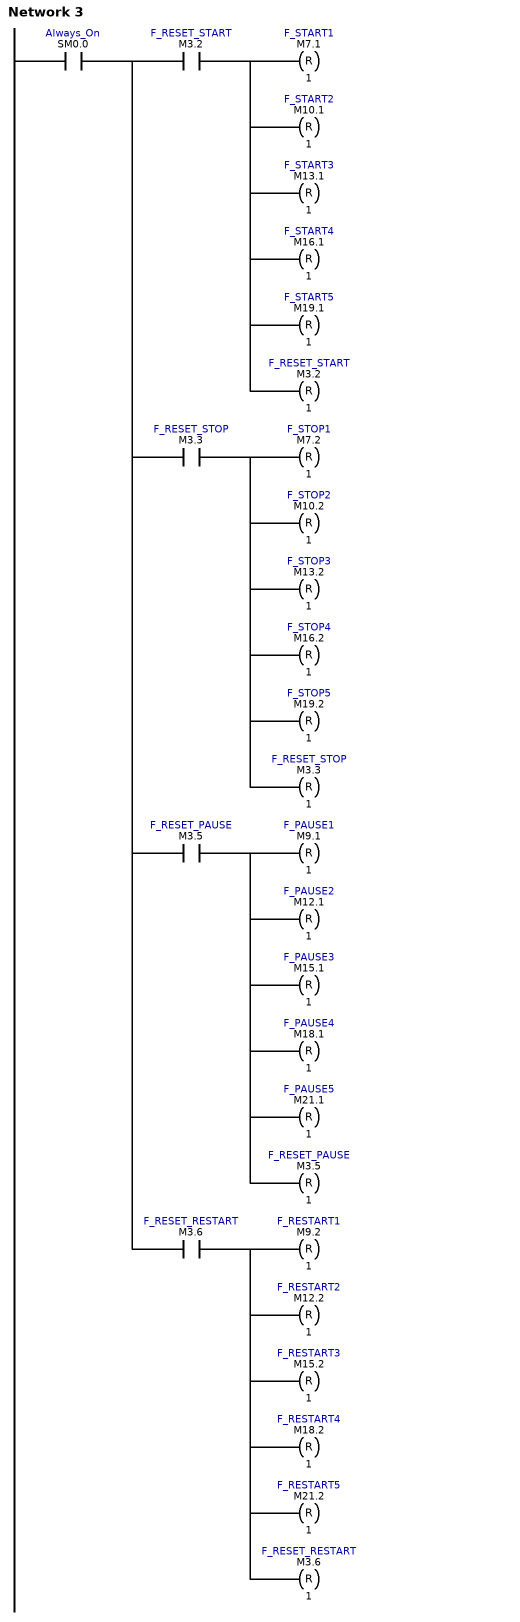
Network 3
LD     Always_On:SM0.0
LPS
A      F_RESET_START:M3.2
R      F_START1:M7.1, 1
R      F_START2:M10.1, 1
R      F_START3:M13.1, 1
R      F_START4:M16.1, 1
R      F_START5:M19.1, 1
R      F_RESET_START:M3.2, 1
LRD
A      F_RESET_STOP:M3.3
R      F_STOP1:M7.2, 1
R      F_STOP2:M10.2, 1
R      F_STOP3:M13.2, 1
R      F_STOP4:M16.2, 1
R      F_STOP5:M19.2, 1
R      F_RESET_STOP:M3.3, 1
LRD
A      F_RESET_PAUSE:M3.5
R      F_PAUSE1:M9.1, 1
R      F_PAUSE2:M12.1, 1
R      F_PAUSE3:M15.1, 1
R      F_PAUSE4:M18.1, 1
R      F_PAUSE5:M21.1, 1
R      F_RESET_PAUSE:M3.5, 1
LPP
A      F_RESET_RESTART:M3.6
R      F_RESTART1:M9.2, 1
R      F_RESTART2:M12.2, 1
R      F_RESTART3:M15.2, 1
R      F_RESTART4:M18.2, 1
R      F_RESTART5:M21.2, 1
R      F_RESET_RESTART:M3.6, 1
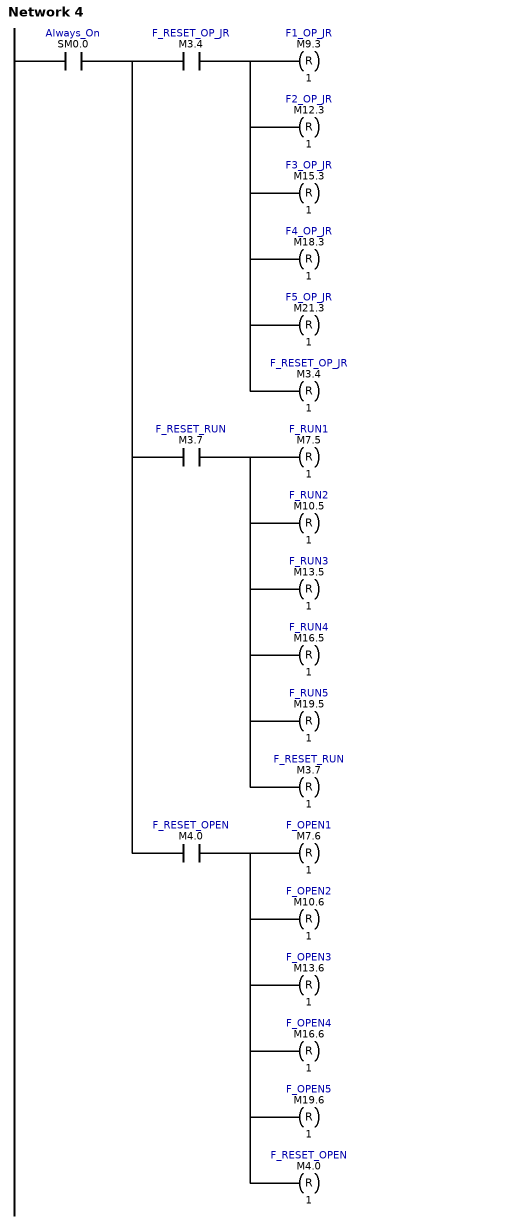
Network 4
LD     Always_On:SM0.0
LPS
A      F_RESET_OP_JR:M3.4
R      F1_OP_JR:M9.3, 1
R      F2_OP_JR:M12.3, 1
R      F3_OP_JR:M15.3, 1
R      F4_OP_JR:M18.3, 1
R      F5_OP_JR:M21.3, 1
R      F_RESET_OP_JR:M3.4, 1
LRD
A      F_RESET_RUN:M3.7
R      F_RUN1:M7.5, 1
R      F_RUN2:M10.5, 1
R      F_RUN3:M13.5, 1
R      F_RUN4:M16.5, 1
R      F_RUN5:M19.5, 1
R      F_RESET_RUN:M3.7, 1
LPP
A      F_RESET_OPEN:M4.0
R      F_OPEN1:M7.6, 1
R      F_OPEN2:M10.6, 1
R      F_OPEN3:M13.6, 1
R      F_OPEN4:M16.6, 1
R      F_OPEN5:M19.6, 1
R      F_RESET_OPEN:M4.0, 1
